//{attribute 'qualified_only'}
//{attribute 'strict'}
TYPE E_Mode :
(
	Mode_Manual := 0,
    Mode_Auto   := 1
);
END_TYPE

(* stored: Version 1.1.0.1, ProductVersion 3.1.4024.15
   DUT E_Mode: Id {f209f172-8f20-4d2a-9c10-7c5eaf2d63ef} *)
